SYSTEM Simple2
  (* Version 1.0, 2019-10-21, badger *)
  APPLICATION Simple2App
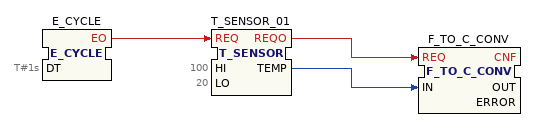
    FBS
      E_CYCLE : E_CYCLE(DT := T#1s);
      T_SENSOR_01 : T_SENSOR(HI := 100, LO := 20);
      F_TO_C_CONV : F_TO_C_CONV;
    END_FBS
    EVENT_CONNECTIONS
      E_CYCLE.EO TO T_SENSOR_01.REQ;
      T_SENSOR_01.REQO TO F_TO_C_CONV.REQ;
    END_CONNECTIONS
    DATA_CONNECTIONS
      T_SENSOR_01.TEMP TO F_TO_C_CONV.IN;
    END_CONNECTIONS
  END_APPLICATION
  DEVICE FORTE_PC : FORTE_PC(MGR_ID := "localhost:61499")
    {SET_ATTRIBUTE(Profile, HOLOBLOC)} (* device profile *)
    RESOURCE EMB_RES : EMB_RES
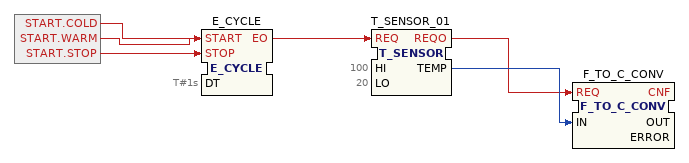
      FBS
        E_CYCLE : E_CYCLE(DT := T#1s);
        T_SENSOR_01 : T_SENSOR(HI := 100, LO := 20);
        F_TO_C_CONV : F_TO_C_CONV;
      END_FBS
      EVENT_CONNECTIONS
        E_CYCLE.EO TO T_SENSOR_01.REQ;
        START.COLD TO E_CYCLE.START;
        START.WARM TO E_CYCLE.START;
        START.STOP TO E_CYCLE.STOP;
        T_SENSOR_01.REQO TO F_TO_C_CONV.REQ;
      END_CONNECTIONS
      DATA_CONNECTIONS
        T_SENSOR_01.TEMP TO F_TO_C_CONV.IN;
      END_CONNECTIONS
    END_RESOURCE
  END_DEVICE
  MAPPINGS
    Simple2App.E_CYCLE ON FORTE_PC.EMB_RES.E_CYCLE;
    Simple2App.T_SENSOR_01 ON FORTE_PC.EMB_RES.T_SENSOR_01;
    Simple2App.F_TO_C_CONV ON FORTE_PC.EMB_RES.F_TO_C_CONV;
  END_MAPPINGS
  SEGMENTS
    Ethernet : Ethernet;
  END_SEGMENTS
  LINKS
    FORTE_PC => Ethernet;
  END_LINKS
END_SYSTEM
